FUNCTION_BLOCK CSVLogger IMPLEMENTS EventLogger
VAR_INPUT
END_VAR
VAR_OUTPUT
END_VAR
VAR
  _path: STRING(255);
  file: TcExt.FileMemory := (mode_write := Tc2_System.FOPEN_MODEAPPEND OR Tc2_System.FOPEN_MODETEXT);
  _done: BOOL;
  _level: EventLevel;
  act_time: TIMESTRUCT;
  format_string: FB_FormatSTring;
  message_queue: FB_FrameFifo;
  state_number: INT;
END_VAR

METHOD INTERNAL create_row : STRING(255)
VAR_INPUT
  ev: EventMessage;
END_VAR
VAR
  dtstr: STRING(255);
  clearedstr: STRING(255);
  levelstr: STRING(255);
END_VAR
IF ev.cleared THEN
  dtstr := TIMESTRUCT_TO_DATETIMESTR(ev.timestamp_cleared);
ELSE
  dtstr := TIMESTRUCT_TO_DATETIMESTR(ev.timestamp_raised);
END_IF
clearedstr := TO_STRING(ev.cleared);
levelstr := TO_STRING(ev.level);

format_string(
  sFormat:='%s,%s,%s,%s,%s$R',
  arg1:=F_STRING(dtstr),
  arg2:=F_STRING(clearedstr),
  arg3:=F_STRING(levelstr),
  arg4:=F_STRING(ev.path),
  arg5:=F_STRING(ev.message),
  sOut=>create_row
);
END_METHOD

METHOD PRIVATE get_timestamped_filename : STRING(255)
VAR
  datestr: STRING(255);
END_VAR
datestr := TIMESTRUCT_TO_DATESTR(act_time);
format_string(
  sFormat:='log_%s.csv',
  arg1:=F_STRING(datestr),
  sOut=>get_timestamped_filename);
END_METHOD

PROPERTY PUBLIC level : EventLevel
GET
level := _level;
END_GET
SET
_level := level;
END_SET
END_PROPERTY

PROPERTY PUBLIC path : STRING(255)
GET
path := _path;
END_GET
SET
_path := path;
END_SET
END_PROPERTY

METHOD run
VAR_INPUT
  act_time: TIMESTRUCT;
END_VAR
THIS^.act_time := act_time;

save();
END_METHOD

METHOD PRIVATE save
VAR
  done: BOOL;
  error_id: DWORD;
END_VAR
CASE state_number OF
0:
  message_queue.RemoveHead();
  IF message_queue.bOk THEN
    file.path := CONCAT(path, get_timestamped_filename());
    file.write(
      start:=FALSE,
      data_ptr:=ADR(message_queue.sGet),
      data_size:=TO_UDINT(LEN(message_queue.sGet))
    );
    state_number := state_number + 10;
	END_IF
10:
  file.write(
    start:=TRUE,
    data_ptr:=ADR(message_queue.sGet),
    data_size:=TO_UDINT(LEN(message_queue.sGet)),
    done=>done,
    error_id=>error_id
  );
  state_number := state_number + 10;
20:
  file.write(
    start:=FALSE,
    data_ptr:=ADR(message_queue.sGet),
    data_size:=TO_UDINT(LEN(message_queue.sGet)),
    done=>done,
    error_id=>error_id
  );
  
  IF done THEN
    state_number := 0;
	END_IF
END_CASE
END_METHOD

METHOD submit_event_message
VAR_IN_OUT
	ev: EventMessage;
END_VAR
IF ev.level >= level THEN
  message_queue.bLog := FALSE;
  message_queue.sPrefix := 'CSVLogger::';
  message_queue.sPut := create_row(ev);
  message_queue.AddTail();
END_IF
END_METHOD

END_FUNCTION_BLOCK

(* stored: Version 1.1.0.1, ProductVersion 3.1.4024.9
   POU CSVLogger: Id {eddd5bf2-9f8b-4014-b1a1-2b9514f6af17}, SpecialFunc None
   Method create_row: Id {62ac12fa-3bef-45d6-b92a-39ca0590c04e}
   Method get_timestamped_filename: Id {fd365ee7-137c-43d5-b097-a6c91d56c64b}
   Property level: Id {ab6b9969-76e1-4879-b617-99481726f092}
   Get Get: Id {5ab1af13-9930-49f3-9811-710132aa1fb1}
   Set Set: Id {cf7d265b-a08f-46d3-959d-33b6de9e6222}
   Property path: Id {8ad77a76-a7ae-4211-a029-62cbfb7f3a1a}
   Get Get: Id {32fab473-3ae0-4d2e-b9ac-c6915164202f}
   Set Set: Id {b4db1cae-d219-49b1-923d-846a377b7031}
   Method run: Id {90c25d9f-9ec4-40ba-a160-c50bc84f515f}
   Method save: Id {501c7d54-f5c2-48f2-862f-f63db1339f45}
   Method submit_event_message: Id {4532367b-994f-48dd-829f-58c767e7db29} *)
